Fanuc KAREL source: kd00039.KL

-- PROVISIONAL review KL for V1013-1; original PC SHA256 1884bab0676e58e84a3bac97b8b445b94d1bc503fd1417dadb4c7a7c1971cff1
-- Incomplete behavior may be omitted. Consult companion uncertainty JSON. Do not deploy.
PROGRAM KD00039
%NOLOCKGROUP
VAR
  I : INTEGER
  J : INTEGER
  B : BOOLEAN
  R : REAL
  S : STRING[80]
BEGIN
  -- UNRESOLVED_PC offsets 5-18; opcodes 9D,81,18,9D,1B,9D,12,9D,13,04
  -- UNRESOLVED_PC offsets 23-27; opcodes 7F
END KD00039
